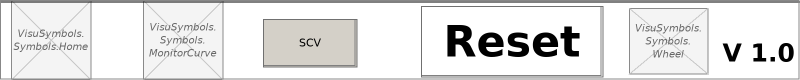
VISUALIZATION Control_Panel  // 800x80
    Image (11,0 80x80), image: VisuSymbols.Symbols.Home
        OnMouseClick: change screen: Overview_ATP
    Image (143,0 80x80), image: VisuSymbols.Symbols.MonitorCurve
        OnMouseClick: change screen: Graph
    Button (421,6 182x71), "Reset"
        tap GVL_IO.Reset
    Line (800,2) (0,2)
    Image (629,8 79x66), image: VisuSymbols.Symbols.Wheel
        OnMouseClick: change screen: Password
    Button (263,19 94x48), "SCV"
        tap GVL_IO.OpenExplorer_cmd
    Label (722,33 74x39), "V 1.0"
END_VISUALIZATION

(* stored: Version 1.1.0.1, ProductVersion 3.1.4024.13
   Visu Control_Panel: Id {d1ba7981-a4e0-4872-910a-eaa15cf20fc1} *)
